KUKA KRL data list: GEOMETRY.dat

&ACCESS RV1
DEFDAT GEOMETRY PUBLIC
   GLOBAL STRUC PLANE3D_T VECTOR3_T P, VECTOR3_T N
   GLOBAL STRUC POSE3D_T VECTOR3_T TRANSLATION, MATRIX3_T ROTATION
ENDDAT
